TYPE ST_Event :
STRUCT
	eEventType: E_EventType;
	eEventSeverity: TcEventSeverity;
	nEventIdentity: UDINT;
	sEventText: STRING(255);
	dtTimeStamp: DT;
END_STRUCT
END_TYPE

(* stored: Version 1.1.0.1, ProductVersion 3.1.4024.11
   DUT ST_Event: Id {b1e2d5f4-2846-44b4-a6a3-15fe8d70bd99} *)
